FUNCTION_BLOCK FB_LamparaTemporizada_SFC_2
// Lampara temporizada con tiempo de espera prolongado
VAR_INPUT
    TiempoEncendido: TIME := T#2S;
    IncrementoTiempo: TIME := T#1S;
END_VAR
VAR_OUTPUT
    TiempoPendiente: REAL;
END_VAR
VAR
    Lampara AT %Q*: BOOL;
    Pulsador AT %I*: BOOL;
END_VAR

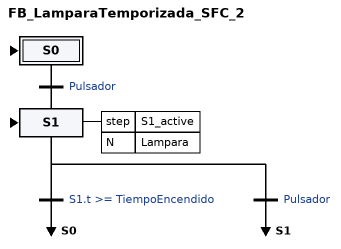
INITIAL_STEP S0:
END_STEP
TRANSITION FROM S0 TO S1
    := Pulsador;
END_TRANSITION
STEP S1:
    S1_active(N);  // step action
    Lampara(N);
END_STEP
TRANSITION FROM S1 TO S0
    := S1.t >= TiempoEncendido;
END_TRANSITION
TRANSITION FROM S1 TO S1
    := Pulsador;
END_TRANSITION

ACTION S1_active:
TiempoPendiente := TiempoEncendido - (TIME_TO_REAL(S1.t)/1000);
END_ACTION

END_FUNCTION_BLOCK

(* stored: Version 1.1.0.1, ProductVersion 3.1.4024.15
   POU FB_LamparaTemporizada_SFC_2: Id {1b2603f0-dd9b-4b51-9d0b-1c3c88b82239}, SpecialFunc None
   Action S1_active: Id {8c1dae8b-8d82-4667-9fe1-df21a82429c1} *)
